(* PLC project average_5, Dassault Systèmes ControlBuild 2024x *)
(* stored: creationDateTime 2023-10-03T11:13:26-01:00 *)

(* This module returns a real. This real corresponds to the average value of real inputs. Number of inputs can go from 2 to 5. *)
FUNCTION_BLOCK equipment_library.average_5
  VAR_INPUT
    input1 : REAL := 0.0;
    input2 : REAL := 0.0;
    input3 : REAL := 0.0;
    input4 : REAL := 0.0;
    input5 : REAL := 0.0;
  END_VAR
  VAR_OUTPUT
    result : REAL := 0.0;
  END_VAR
  VAR CONSTANT
    nbInputs : DINT := 2;
  END_VAR
  VAR
    d_average : BOOL := false;
    v_d_average : REAL := 0.0;
  END_VAR


ACTION C_source_code:
/* ----------------------------------------------------------------	*/
/* Type : Model of Operative Behaviour					*/
/* Category :  Toolbox							*/
/* Author : Dassault Systemes						*/
/* Update date : June 2018						*/
/* ----------------------------------------------------------------	*/
/* This module returns a real. 						*/
/* This real corresponds to the average value of real inputs.		*/
/* Number of inputs can gone from 2 to 5. 				*/
/* ----------------------------------------------------------------	*/

if (d_average) result = v_d_average;
else {
	switch(nbInputs) {
		case 2 : result = input1 + input2;
			break;
		case 3 : result = input1 + input2 + input3;
			break;
		case 4 : result = input1 + input2 + input3 + input4;
			break;
		case 5 : result = input1 + input2 + input3 + input4 + input5; 
			break;
		default : result = 0.0;
		
			break;
	}

	if (nbInputs > 0) result = result / nbInputs;
}
END_ACTION
END_FUNCTION_BLOCK
